--- program Path2 (robot UR5) ---
  Smooth(1)
  Set Ref.: Frame 2 at (-32.2, -480, 0) mm
  Set Tool: laser_fixture_tool
  Show laser_fixture_tool
  Set speed (1000.0 mm/s)
  MoveJ 1 to (-97.68, -19.69, 50.49) mm, rotated rx -95.37 ry 46.1 rz -97.44 deg; joints [-117.398, -152.62, -79.729, 61.497, 204.11, 54.589]
  MoveL 2 to (-97.68, -19.69, 50.49) mm, rotated rx -95.37 ry 46.1 rz -97.44 deg; joints [-117.398, -152.62, -79.729, 61.497, 204.11, 54.589]
  MoveL 3 to (1.91, -25.89, 44) mm, rotated rx -95.37 ry 46.1 rz -97.44 deg; joints [-108.024, -149.891, -88.195, 72.69, 194.926, 60.358]
  MoveL 4 to (1.91, -25.89, 44) mm, rotated rx -95.37 ry 46.1 rz -97.44 deg; joints [-108.024, -149.891, -88.195, 72.69, 194.926, 60.358]
  Set speed (100.0 mm/s)
  MoveL 5 to (1.98, -24.59, 43.9) mm, rotated rx -94.01 ry 38.49 rz -96.43 deg; joints [-108.115, -149.874, -89.181, 71.68, 194.519, 50.789]
  MoveL 6 to (2.06, -23.31, 43.74) mm, rotated rx -92.48 ry 28.02 rz -95.27 deg; joints [-108.188, -149.973, -90.447, 69.355, 194.248, 36.704]
  MoveL 7 to (2.12, -22.3, 43.59) mm, rotated rx -91.26 ry 16 rz -94.57 deg; joints [-108.24, -150.074, -91.694, 66.761, 194.073, 20.852]
  MoveL 8 to (2.19, -21.29, 43.41) mm, rotated rx -90.07 ry 0.97 rz -94.25 deg; joints [-108.275, -150.182, -93.079, 63.558, 194.03, 1.259]
  MoveL 9 to (2.26, -20.27, 43.2) mm, rotated rx -88.73 ry -16.32 rz -94.53 deg; joints [-108.287, -150.286, -94.55, 59.834, 194.17, -21.172]
  MoveL 10 to (2.33, -19.25, 42.96) mm, rotated rx -86.87 ry -33.13 rz -95.71 deg; joints [-108.274, -150.382, -96, 55.867, 194.507, -43.358]
  MoveL 11 to (2.41, -18.24, 42.7) mm, rotated rx -83.97 ry -47.18 rz -98.2 deg; joints [-108.236, -150.476, -97.37, 51.853, 195.027, -62.813]
  MoveL 12 to (2.5, -17.15, 42.4) mm, rotated rx -78.9 ry -58.66 rz -102.94 deg; joints [-108.162, -150.604, -98.668, 47.676, 195.795, -79.986]
  MoveL 13 to (2.6, -15.98, 42.05) mm, rotated rx -70.11 ry -67.29 rz -111.42 deg; joints [-108.046, -150.804, -99.778, 43.597, 196.83, -94.499]
  MoveL 14 to (2.71, -14.82, 41.67) mm, rotated rx -56.63 ry -72.85 rz -124.58 deg; joints [-107.893, -151.088, -100.576, 40.065, 198.034, -105.875]
  MoveL 15 to (2.81, -13.7, 41.29) mm, rotated rx -39.3 ry -75.67 rz -141.58 deg; joints [-107.714, -151.441, -101.097, 37.153, 199.307, -114.647]
  MoveL 16 to (2.92, -12.62, 40.89) mm, rotated rx -21.62 ry -76.38 rz -158.93 deg; joints [-107.516, -151.847, -101.404, 34.774, 200.599, -121.547]
  MoveL 17 to (3.02, -11.55, 40.47) mm, rotated rx -6.64 ry -75.69 rz -173.56 deg; joints [-107.294, -152.307, -101.552, 32.769, 201.93, -127.281]
  MoveL 18 to (3.14, -10.42, 40.01) mm, rotated rx 5.46 ry -74.12 rz 174.75 deg; joints [-107.034, -152.855, -101.524, 31.037, 203.383, -132.45]
  MoveL 19 to (3.26, -9.3, 39.53) mm, rotated rx 13.98 ry -72.1 rz 166.68 deg; joints [-106.75, -153.449, -101.357, 29.617, 204.857, -136.867]
  MoveL 20 to (3.38, -8.19, 39.02) mm, rotated rx 20.16 ry -69.89 rz 160.98 deg; joints [-106.442, -154.081, -101.056, 28.479, 206.349, -140.71]
  MoveL 21 to (3.5, -7.16, 38.53) mm, rotated rx 24.31 ry -67.77 rz 157.31 deg; joints [-106.138, -154.692, -100.702, 27.595, 207.742, -143.855]
  MoveL 22 to (3.62, -6.13, 38.01) mm, rotated rx 27.45 ry -65.69 rz 154.67 deg; joints [-105.824, -155.305, -100.283, 26.893, 209.104, -146.603]
  MoveL 23 to (3.74, -5.11, 37.48) mm, rotated rx 29.93 ry -63.69 rz 152.7 deg; joints [-105.508, -155.909, -99.812, 26.36, 210.414, -148.998]
  MoveL 24 to (3.87, -4.1, 36.93) mm, rotated rx 31.98 ry -61.8 rz 151.18 deg; joints [-105.197, -156.492, -99.304, 25.985, 211.65, -151.075]
  MoveL 25 to (3.99, -3.1, 36.36) mm, rotated rx 33.74 ry -60.04 rz 149.95 deg; joints [-104.899, -157.044, -98.773, 25.755, 212.794, -152.865]
  MoveL 26 to (4.12, -2.14, 35.78) mm, rotated rx 35.25 ry -58.46 rz 148.94 deg; joints [-104.624, -157.546, -98.249, 25.647, 213.814, -154.372]
  MoveL 27 to (4.25, -1.18, 35.18) mm, rotated rx 36.76 ry -56.98 rz 147.94 deg; joints [-104.37, -158.013, -97.693, 25.681, 214.733, -155.685]
  MoveL 28 to (4.37, -0.31, 34.6) mm, rotated rx 38.13 ry -55.7 rz 147.04 deg; joints [-104.155, -158.41, -97.17, 25.81, 215.493, -156.743]
  MoveL 29 to (4.5, 0.55, 34.01) mm, rotated rx 39.62 ry -54.47 rz 146.03 deg; joints [-103.959, -158.78, -96.605, 26.059, 216.174, -157.692]
  MoveL 30 to (4.62, 1.39, 33.4) mm, rotated rx 41.27 ry -53.25 rz 144.88 deg; joints [-103.782, -159.123, -95.99, 26.432, 216.78, -158.557]
  MoveL 31 to (4.74, 2.19, 32.8) mm, rotated rx 42.33 ry -52.31 rz 144.22 deg; joints [-103.635, -159.404, -95.553, 26.685, 217.275, -159.223]
  MoveL 32 to (4.91, 3.31, 31.9) mm, rotated rx 44.8 ry -50.73 rz 142.45 deg; joints [-103.451, -159.789, -94.649, 27.444, 217.892, -160.186]
  MoveL 33 to (5.08, 4.4, 30.96) mm, rotated rx 47.43 ry -49.14 rz 140.54 deg; joints [-103.305, -160.117, -93.707, 28.355, 218.378, -161.045]
  MoveL 34 to (5.25, 5.45, 29.99) mm, rotated rx 49.49 ry -47.83 rz 139.06 deg; joints [-103.198, -160.376, -92.96, 29.156, 218.736, -161.713]
  MoveL 35 to (5.43, 6.44, 28.99) mm, rotated rx 50.93 ry -46.84 rz 138.05 deg; joints [-103.118, -160.586, -92.43, 29.783, 218.999, -162.207]
  MoveL 36 to (5.61, 7.35, 28) mm, rotated rx 51.83 ry -46.14 rz 137.47 deg; joints [-103.051, -160.768, -92.087, 30.223, 219.211, -162.569]
  MoveL 37 to (5.8, 8.16, 27.05) mm, rotated rx 52.21 ry -45.7 rz 137.3 deg; joints [-102.985, -160.938, -91.909, 30.456, 219.407, -162.832]
  MoveL 38 to (6.01, 8.91, 26.1) mm, rotated rx 52.19 ry -45.41 rz 137.45 deg; joints [-102.907, -161.118, -91.833, 30.519, 219.628, -163.057]
  MoveL 39 to (6.25, 9.59, 25.16) mm, rotated rx 51.89 ry -45.19 rz 137.87 deg; joints [-102.804, -161.322, -91.806, 30.444, 219.904, -163.292]
  MoveL 40 to (6.49, 10.19, 24.25) mm, rotated rx 51.29 ry -45.01 rz 138.58 deg; joints [-102.671, -161.555, -91.827, 30.209, 220.257, -163.553]
  MoveL 41 to (6.77, 10.75, 23.33) mm, rotated rx 50.5 ry -44.77 rz 139.49 deg; joints [-102.494, -161.833, -91.835, 29.864, 220.718, -163.892]
  MoveL 42 to (7.09, 11.26, 22.39) mm, rotated rx 49.64 ry -44.4 rz 140.54 deg; joints [-102.268, -162.162, -91.794, 29.446, 221.298, -164.331]
  MoveL 43 to (7.44, 11.72, 21.44) mm, rotated rx 48.8 ry -43.88 rz 141.63 deg; joints [-101.995, -162.534, -91.675, 28.993, 221.99, -164.871]
  MoveL 44 to (7.81, 12.11, 20.53) mm, rotated rx 48.83 ry -43.04 rz 142.03 deg; joints [-101.733, -162.885, -91.275, 28.886, 222.626, -165.478]
  MoveL 45 to (7.95, 12.23, 20.22) mm, rotated rx 49.41 ry -42.62 rz 141.68 deg; joints [-101.675, -162.97, -90.985, 29.096, 222.751, -165.687]
  Set speed (1000.0 mm/s)
  MoveL 46 to (7.95, 12.23, 20.22) mm, rotated rx 49.41 ry -42.62 rz 141.68 deg; joints [-101.675, -162.97, -90.985, 29.096, 222.751, -165.687]
  MoveL 47 to (-73.7, -20.03, -27.66) mm, rotated rx 49.41 ry -42.62 rz 141.68 deg; joints [-108.268, -173.052, -72.375, 25.011, 227.608, -159.391]
  Set speed (1000.0 mm/s)
  MoveL 48 to (-97.55, 35.36, 42.52) mm, rotated rx -88.89 ry -10.51 rz -96.06 deg; joints [-120.475, -150.967, -92.517, 60.869, 204.643, -12.887]
  MoveL 49 to (1.91, 25.16, 44.42) mm, rotated rx -88.89 ry -10.51 rz -96.06 deg; joints [-110.164, -147.723, -102.71, 66.031, 194.349, -14.776]
  MoveL 50 to (1.91, 25.16, 44.42) mm, rotated rx -88.89 ry -10.51 rz -96.06 deg; joints [-110.164, -147.723, -102.71, 66.031, 194.349, -14.776]
  Set speed (100.0 mm/s)
  MoveL 51 to (1.98, 25.72, 43.25) mm, rotated rx -88.19 ry -17.29 rz -96.08 deg; joints [-110.132, -148.034, -103.098, 64.289, 194.692, -23.923]
  MoveL 52 to (2.06, 26.23, 42.05) mm, rotated rx -87.4 ry -25.95 rz -95.93 deg; joints [-110.04, -148.436, -103.065, 62.671, 195.424, -34.491]
  MoveL 53 to (2.12, 26.6, 41.1) mm, rotated rx -86.33 ry -36.31 rz -96.18 deg; joints [-109.931, -148.826, -102.954, 61.128, 196.192, -46.606]
  MoveL 54 to (2.19, 26.95, 40.14) mm, rotated rx -84.48 ry -49.54 rz -97.24 deg; joints [-109.789, -149.268, -102.655, 59.677, 197.122, -61.387]
  MoveL 55 to (2.26, 27.27, 39.15) mm, rotated rx -79.85 ry -65.51 rz -101.13 deg; joints [-109.61, -149.762, -102.145, 58.387, 198.206, -78.71]
  MoveL 56 to (2.33, 27.58, 38.15) mm, rotated rx -55.43 ry -81.59 rz -124.86 deg; joints [-109.399, -150.29, -101.463, 57.275, 199.392, -96.746]
  MoveL 57 to (2.41, 27.86, 37.15) mm, rotated rx 58.45 ry -79.77 rz 121.96 deg; joints [-109.16, -150.846, -100.674, 56.248, 200.649, -113.072]
  MoveL 58 to (2.5, 28.14, 36.05) mm, rotated rx 74.81 ry -66.9 rz 106.44 deg; joints [-108.873, -151.466, -99.702, 55.284, 202.062, -127.151]
  MoveL 59 to (2.6, 28.42, 34.87) mm, rotated rx 78.42 ry -56.07 rz 103.87 deg; joints [-108.537, -152.135, -98.547, 54.435, 203.605, -138.342]
  MoveL 60 to (2.71, 28.68, 33.67) mm, rotated rx 79.75 ry -47.86 rz 103.7 deg; joints [-108.18, -152.789, -97.305, 53.779, 205.14, -146.526]
  MoveL 61 to (2.81, 28.9, 32.51) mm, rotated rx 80.34 ry -41.76 rz 104.33 deg; joints [-107.819, -153.406, -96.068, 53.252, 206.603, -152.411]
  MoveL 62 to (2.92, 29.1, 31.38) mm, rotated rx 80.63 ry -37.16 rz 105.29 deg; joints [-107.46, -153.987, -94.871, 52.799, 207.986, -156.733]
  MoveL 63 to (3.02, 29.28, 30.24) mm, rotated rx 80.77 ry -33.45 rz 106.42 deg; joints [-107.092, -154.551, -93.682, 52.386, 209.335, -160.107]
  MoveL 64 to (3.14, 29.44, 29.03) mm, rotated rx 80.98 ry -29.94 rz 107.64 deg; joints [-106.696, -155.114, -92.391, 52.087, 210.724, -163.092]
  MoveL 65 to (3.26, 29.58, 27.82) mm, rotated rx 81.2 ry -26.87 rz 108.91 deg; joints [-106.294, -155.65, -91.099, 51.853, 212.077, -165.555]
  MoveL 66 to (3.38, 29.7, 26.61) mm, rotated rx 81.49 ry -24.03 rz 110.17 deg; joints [-105.888, -156.149, -89.791, 51.726, 213.39, -167.677]
  MoveL 67 to (3.5, 29.79, 25.46) mm, rotated rx 81.76 ry -21.7 rz 111.4 deg; joints [-105.504, -156.6, -88.587, 51.615, 214.592, -169.337]
  MoveL 68 to (3.62, 29.86, 24.31) mm, rotated rx 82.05 ry -19.58 rz 112.61 deg; joints [-105.124, -157.021, -87.412, 51.55, 215.741, -170.757]
  MoveL 69 to (3.74, 29.91, 23.17) mm, rotated rx 82.39 ry -17.66 rz 113.77 deg; joints [-104.756, -157.407, -86.281, 51.538, 216.822, -171.975]
  MoveL 70 to (3.87, 29.93, 22.02) mm, rotated rx 82.78 ry -15.88 rz 114.85 deg; joints [-104.406, -157.754, -85.205, 51.582, 217.821, -173.027]
  MoveL 71 to (3.99, 29.93, 20.87) mm, rotated rx 83.21 ry -14.24 rz 115.84 deg; joints [-104.082, -158.056, -84.199, 51.692, 218.723, -173.941]
  MoveL 72 to (4.12, 29.91, 19.74) mm, rotated rx 83.63 ry -12.81 rz 116.73 deg; joints [-103.789, -158.322, -83.295, 51.823, 219.514, -174.697]
  MoveL 73 to (4.25, 29.87, 18.61) mm, rotated rx 84.14 ry -11.38 rz 117.48 deg; joints [-103.53, -158.531, -82.452, 52.062, 220.197, -175.401]
  MoveL 74 to (4.37, 29.81, 17.57) mm, rotated rx 84.59 ry -10.22 rz 118.11 deg; joints [-103.314, -158.707, -81.751, 52.28, 220.752, -175.949]
  MoveL 75 to (4.5, 29.73, 16.53) mm, rotated rx 85.11 ry -9.02 rz 118.63 deg; joints [-103.127, -158.835, -81.096, 52.592, 221.22, -176.485]
  MoveL 76 to (4.62, 29.62, 15.5) mm, rotated rx 85.75 ry -7.69 rz 119.02 deg; joints [-102.972, -158.905, -80.479, 53.039, 221.596, -177.042]
  MoveL 77 to (4.74, 29.5, 14.5) mm, rotated rx 85.8 ry -7.44 rz 119.58 deg; joints [-102.802, -159.131, -80.043, 52.942, 222.007, -177.183]
  MoveL 78 to (4.91, 29.28, 13.09) mm, rotated rx 86.75 ry -5.66 rz 119.88 deg; joints [-102.658, -159.144, -79.34, 53.684, 222.322, -177.88]
  MoveL 79 to (5.08, 29.01, 11.67) mm, rotated rx 87.98 ry -3.51 rz 119.97 deg; joints [-102.577, -159.024, -78.704, 54.74, 222.463, -178.695]
  MoveL 80 to (5.25, 28.69, 10.28) mm, rotated rx 89.05 ry -1.64 rz 120.03 deg; joints [-102.522, -158.914, -78.188, 55.701, 222.53, -179.393]
  MoveL 81 to (5.43, 28.33, 8.92) mm, rotated rx 89.88 ry -0.2 rz 120.1 deg; joints [-102.475, -158.856, -77.771, 56.457, 222.571, -179.927]
  MoveL 82 to (5.61, 27.93, 7.64) mm, rotated rx 90.48 ry 0.83 rz 120.2 deg; joints [-102.423, -158.862, -77.418, 56.992, 222.62, -180.305]
  MoveL 83 to (5.8, 27.51, 6.46) mm, rotated rx 90.82 ry 1.4 rz 120.38 deg; joints [-102.35, -158.951, -77.096, 57.254, 222.721, -180.511]
  MoveL 84 to (6.01, 27.06, 5.34) mm, rotated rx 90.99 ry 1.67 rz 120.66 deg; joints [-102.25, -159.104, -76.764, 57.323, 222.886, -180.606]
  MoveL 85 to (6.25, 26.58, 4.28) mm, rotated rx 91.07 ry 1.79 rz 121.02 deg; joints [-102.12, -159.301, -76.395, 57.266, 223.122, -180.64]
  MoveL 86 to (6.49, 26.1, 3.3) mm, rotated rx 91.01 ry 1.65 rz 121.54 deg; joints [-101.946, -159.565, -75.976, 57.014, 223.47, -180.583]
  MoveL 87 to (6.77, 25.58, 2.36) mm, rotated rx 90.92 ry 1.46 rz 122.22 deg; joints [-101.725, -159.869, -75.473, 56.67, 223.927, -180.506]
  MoveL 88 to (7.09, 25.02, 1.44) mm, rotated rx 90.84 ry 1.3 rz 123.04 deg; joints [-101.459, -160.198, -74.88, 56.28, 224.49, -180.438]
  MoveL 89 to (7.44, 24.43, 0.58) mm, rotated rx 90.81 ry 1.21 rz 124 deg; joints [-101.151, -160.532, -74.203, 55.884, 225.142, -180.397]
  MoveL 90 to (7.81, 23.83, -0.22) mm, rotated rx 91.3 ry 1.88 rz 124.66 deg; joints [-100.929, -160.632, -73.599, 56.053, 225.559, -180.608]
  MoveL 91 to (7.95, 23.62, -0.48) mm, rotated rx 91.81 ry 2.62 rz 124.61 deg; joints [-100.934, -160.496, -73.485, 56.516, 225.491, -180.847]
  Set speed (1000.0 mm/s)
  MoveL 92 to (7.95, 23.62, -0.48) mm, rotated rx 91.81 ry 2.62 rz 124.61 deg; joints [-100.934, -160.496, -73.485, 56.516, 225.491, -180.847]
  MoveL 93 to (-74.39, -33.03, 2.67) mm, rotated rx 91.81 ry 2.62 rz 124.61 deg; joints [-106.621, -168.974, -51.295, 42.589, 231.173, -181.169]
  Set speed (1000.0 mm/s)
  MoveL 94 to (-97.68, 53.58, -8.19) mm, rotated rx -72.98 ry -72.89 rz -107.76 deg; joints [-120.487, -158.48, -90.615, 58.994, 209.415, -82.414]
  MoveL 95 to (1.91, 51.05, 0.42) mm, rotated rx -72.98 ry -72.89 rz -107.76 deg; joints [-110.485, -154.518, -103.068, 62.737, 199.64, -87.613]
  MoveL 96 to (1.91, 51.05, 0.42) mm, rotated rx -72.98 ry -72.89 rz -107.76 deg; joints [-110.485, -154.518, -103.068, 62.737, 199.64, -87.613]
  Set speed (100.0 mm/s)
  MoveL 97 to (1.98, 50.31, -0.65) mm, rotated rx -60.07 ry -79.99 rz -120.31 deg; joints [-110.333, -154.806, -102.376, 62.619, 200.171, -95.008]
  MoveL 98 to (2.06, 49.53, -1.69) mm, rotated rx 22.06 ry -84.98 rz 158.02 deg; joints [-110.154, -155.029, -101.323, 63.16, 200.811, -104.247]
  MoveL 99 to (2.12, 48.9, -2.48) mm, rotated rx 72.87 ry -75.39 rz 107.66 deg; joints [-109.98, -155.191, -100.295, 63.767, 201.447, -114.914]
  MoveL 100 to (2.19, 48.24, -3.26) mm, rotated rx 82.4 ry -60.69 rz 98.7 deg; joints [-109.787, -155.315, -99.138, 64.567, 202.148, -128.264]
  MoveL 101 to (2.26, 47.54, -4.04) mm, rotated rx 85.87 ry -43.48 rz 95.99 deg; joints [-109.575, -155.395, -97.868, 65.545, 202.908, -143.564]
  MoveL 102 to (2.33, 46.83, -4.81) mm, rotated rx 87.6 ry -26.64 rz 95.35 deg; joints [-109.346, -155.428, -96.545, 66.622, 203.71, -158.244]
  MoveL 103 to (2.41, 46.1, -5.55) mm, rotated rx 88.77 ry -12.46 rz 95.7 deg; joints [-109.101, -155.424, -95.197, 67.721, 204.559, -170.17]
  MoveL 104 to (2.5, 45.3, -6.35) mm, rotated rx 89.92 ry -0.69 rz 96.69 deg; joints [-108.819, -155.373, -93.741, 68.926, 205.509, -179.481]
  MoveL 105 to (2.6, 44.41, -7.18) mm, rotated rx 91.24 ry 8.62 rz 98.2 deg; joints [-108.504, -155.267, -92.215, 70.221, 206.544, -186.174]
  MoveL 106 to (2.71, 43.5, -8) mm, rotated rx 92.7 ry 15.52 rz 100 deg; joints [-108.181, -155.111, -90.759, 71.5, 207.574, -190.539]
  MoveL 107 to (2.81, 42.61, -8.78) mm, rotated rx 94.25 ry 20.57 rz 101.95 deg; joints [-107.86, -154.925, -89.421, 72.692, 208.569, -193.276]
  MoveL 108 to (2.92, 41.72, -9.51) mm, rotated rx 95.86 ry 24.37 rz 103.96 deg; joints [-107.544, -154.719, -88.201, 73.792, 209.522, -194.995]
  MoveL 109 to (3.02, 40.83, -10.23) mm, rotated rx 97.55 ry 27.42 rz 106.06 deg; joints [-107.224, -154.491, -87.054, 74.845, 210.466, -196.106]
  MoveL 110 to (3.14, 39.86, -10.98) mm, rotated rx 99.48 ry 30.17 rz 108.37 deg; joints [-106.885, -154.21, -85.922, 75.969, 211.439, -196.911]
  MoveL 111 to (3.26, 38.88, -11.71) mm, rotated rx 101.51 ry 32.49 rz 110.76 deg; joints [-106.544, -153.899, -84.869, 77.078, 212.397, -197.407]
  MoveL 112 to (3.38, 37.89, -12.42) mm, rotated rx 103.67 ry 34.51 rz 113.24 deg; joints [-106.203, -153.549, -83.898, 78.205, 213.333, -197.712]
  MoveL 113 to (3.5, 36.94, -13.07) mm, rotated rx 105.76 ry 36.1 rz 115.6 deg; joints [-105.88, -153.203, -83.052, 79.239, 214.203, -197.823]
  MoveL 114 to (3.62, 35.99, -13.7) mm, rotated rx 107.89 ry 37.46 rz 117.96 deg; joints [-105.562, -152.84, -82.283, 80.256, 215.042, -197.829]
  MoveL 115 to (3.74, 35.01, -14.32) mm, rotated rx 110.03 ry 38.63 rz 120.28 deg; joints [-105.254, -152.466, -81.597, 81.254, 215.836, -197.771]
  MoveL 116 to (3.87, 34.03, -14.91) mm, rotated rx 112.14 ry 39.64 rz 122.52 deg; joints [-104.962, -152.088, -80.998, 82.233, 216.568, -197.681]
  MoveL 117 to (3.99, 33.04, -15.49) mm, rotated rx 114.19 ry 40.52 rz 124.65 deg; joints [-104.693, -151.712, -80.486, 83.185, 217.226, -197.584]
  MoveL 118 to (4.12, 32.05, -16.04) mm, rotated rx 116.12 ry 41.29 rz 126.61 deg; joints [-104.452, -151.356, -80.062, 84.085, 217.793, -197.494]
  MoveL 119 to (4.25, 31.06, -16.56) mm, rotated rx 118.01 ry 42.05 rz 128.46 deg; joints [-104.243, -150.995, -79.727, 84.999, 218.263, -197.458]
  MoveL 120 to (4.37, 30.12, -17.03) mm, rotated rx 119.71 ry 42.73 rz 130.07 deg; joints [-104.077, -150.667, -79.485, 85.842, 218.616, -197.464]
  MoveL 121 to (4.5, 29.18, -17.48) mm, rotated rx 121.44 ry 43.48 rz 131.62 deg; joints [-103.941, -150.324, -79.322, 86.736, 218.878, -197.545]
  MoveL 122 to (4.62, 28.23, -17.9) mm, rotated rx 123.23 ry 44.32 rz 133.16 deg; joints [-103.84, -149.961, -79.242, 87.702, 219.042, -197.713]
  MoveL 123 to (4.74, 27.31, -18.29) mm, rotated rx 124.62 ry 44.85 rz 134.39 deg; joints [-103.737, -149.704, -79.122, 88.405, 219.214, -197.761]
  MoveL 124 to (4.91, 25.97, -18.81) mm, rotated rx 127.16 ry 46.15 rz 136.42 deg; joints [-103.679, -149.19, -79.191, 89.834, 219.202, -198.177]
  MoveL 125 to (5.08, 24.62, -19.29) mm, rotated rx 129.83 ry 47.58 rz 138.48 deg; joints [-103.675, -148.665, -79.374, 91.349, 219.034, -198.729]
  MoveL 126 to (5.25, 23.24, -19.71) mm, rotated rx 132.09 ry 48.72 rz 140.24 deg; joints [-103.675, -148.262, -79.507, 92.588, 218.852, -199.185]
  MoveL 127 to (5.43, 21.89, -20.07) mm, rotated rx 133.83 ry 49.53 rz 141.6 deg; joints [-103.661, -147.994, -79.546, 93.49, 218.711, -199.492]
  MoveL 128 to (5.61, 20.58, -20.37) mm, rotated rx 135.07 ry 50.01 rz 142.61 deg; joints [-103.622, -147.835, -79.488, 94.089, 218.641, -199.638]
  MoveL 129 to (5.8, 19.35, -20.59) mm, rotated rx 135.83 ry 50.18 rz 143.27 deg; joints [-103.551, -147.767, -79.328, 94.4, 218.675, -199.606]
  MoveL 130 to (6.01, 18.15, -20.76) mm, rotated rx 136.28 ry 50.1 rz 143.73 deg; joints [-103.442, -147.751, -79.081, 94.521, 218.817, -199.415]
  MoveL 131 to (6.25, 17, -20.88) mm, rotated rx 136.57 ry 49.83 rz 144.12 deg; joints [-103.296, -147.749, -78.771, 94.534, 219.066, -199.092]
  MoveL 132 to (6.49, 15.91, -20.95) mm, rotated rx 136.73 ry 49.35 rz 144.46 deg; joints [-103.105, -147.757, -78.393, 94.436, 219.449, -198.619]
  MoveL 133 to (6.77, 14.83, -20.97) mm, rotated rx 136.92 ry 48.72 rz 144.9 deg; joints [-102.867, -147.739, -77.968, 94.322, 219.957, -198.032]
  MoveL 134 to (7.09, 13.76, -20.94) mm, rotated rx 137.25 ry 48 rz 145.51 deg; joints [-102.585, -147.671, -77.519, 94.247, 220.579, -197.361]
  MoveL 135 to (7.44, 12.71, -20.87) mm, rotated rx 137.77 ry 47.23 rz 146.33 deg; joints [-102.266, -147.538, -77.077, 94.258, 221.294, -196.645]
  MoveL 136 to (7.81, 11.72, -20.75) mm, rotated rx 138.98 ry 46.94 rz 147.56 deg; joints [-102.021, -147.228, -76.896, 94.747, 221.787, -196.225]
  MoveL 137 to (7.95, 11.39, -20.7) mm, rotated rx 139.78 ry 47.2 rz 148.18 deg; joints [-102.006, -147.032, -77.006, 95.203, 221.761, -196.298]
  Set speed (1000.0 mm/s)
  MoveL 138 to (7.95, 11.39, -20.7) mm, rotated rx 139.78 ry 47.2 rz 148.18 deg; joints [-102.006, -147.032, -77.006, 95.203, 221.761, -196.298]
  MoveL 139 to (-73.7, -13.94, 31.18) mm, rotated rx 139.78 ry 47.2 rz 148.18 deg; joints [-108.931, -148.976, -64.289, 79.063, 226.36, -203.756]
  Set speed (1000.0 mm/s)
  MoveL 140 to (-97.68, 19.69, -50.49) mm, rotated rx 84.63 ry -46.1 rz 97.44 deg; joints [-117.798, -165.768, -78.334, 56.973, 211.556, -139.855]
  MoveL 141 to (1.91, 25.89, -44) mm, rotated rx 84.63 ry -46.1 rz 97.44 deg; joints [-108.738, -161.585, -91.609, 63.461, 202.592, -142.771]
  MoveL 142 to (1.91, 25.89, -44) mm, rotated rx 84.63 ry -46.1 rz 97.44 deg; joints [-108.738, -161.585, -91.609, 63.461, 202.592, -142.771]
  Set speed (100.0 mm/s)
  MoveL 143 to (1.98, 24.59, -43.9) mm, rotated rx 85.99 ry -38.49 rz 96.43 deg; joints [-108.636, -161.508, -90.877, 64.247, 202.775, -148.954]
  MoveL 144 to (2.06, 23.31, -43.74) mm, rotated rx 87.52 ry -28.02 rz 95.27 deg; joints [-108.573, -161.275, -90.128, 65.736, 202.779, -157.189]
  MoveL 145 to (2.12, 22.3, -43.59) mm, rotated rx 88.74 ry -16 rz 94.57 deg; joints [-108.525, -161.003, -89.455, 67.324, 202.774, -166.881]
  MoveL 146 to (2.19, 21.29, -43.41) mm, rotated rx 89.93 ry -0.97 rz 94.25 deg; joints [-108.485, -160.649, -88.774, 69.236, 202.73, -179.201]
  MoveL 147 to (2.26, 20.27, -43.2) mm, rotated rx 91.27 ry 16.32 rz 94.53 deg; joints [-108.451, -160.202, -88.099, 71.478, 202.652, -193.389]
  MoveL 148 to (2.33, 19.25, -42.96) mm, rotated rx 93.13 ry 33.13 rz 95.71 deg; joints [-108.419, -159.674, -87.452, 73.968, 202.564, -206.849]
  MoveL 149 to (2.41, 18.24, -42.7) mm, rotated rx 96.03 ry 47.18 rz 98.2 deg; joints [-108.381, -159.07, -86.83, 76.657, 202.504, -217.387]
  MoveL 150 to (2.5, 17.15, -42.4) mm, rotated rx 101.1 ry 58.66 rz 102.94 deg; joints [-108.333, -158.333, -86.216, 79.744, 202.471, -225.046]
  MoveL 151 to (2.6, 15.98, -42.05) mm, rotated rx 109.89 ry 67.29 rz 111.42 deg; joints [-108.273, -157.452, -85.651, 83.202, 202.477, -229.833]
  MoveL 152 to (2.71, 14.82, -41.67) mm, rotated rx 123.37 ry 72.85 rz 124.58 deg; joints [-108.204, -156.491, -85.203, 86.74, 202.53, -232.203]
  MoveL 153 to (2.81, 13.7, -41.29) mm, rotated rx 140.7 ry 75.67 rz 141.58 deg; joints [-108.123, -155.493, -84.879, 90.193, 202.644, -232.933]
  MoveL 154 to (2.92, 12.62, -40.89) mm, rotated rx 158.38 ry 76.38 rz 158.93 deg; joints [-108.032, -154.475, -84.671, 93.513, 202.818, -232.673]
  MoveL 155 to (3.02, 11.55, -40.47) mm, rotated rx 173.36 ry 75.69 rz 173.56 deg; joints [-107.928, -153.412, -84.567, 96.798, 203.051, -231.796]
  MoveL 156 to (3.14, 10.42, -40.01) mm, rotated rx -174.54 ry 74.12 rz -174.75 deg; joints [-107.81, -152.234, -84.589, 100.273, 203.333, -230.532]
  MoveL 157 to (3.26, 9.3, -39.53) mm, rotated rx -166.02 ry 72.1 rz -166.68 deg; joints [-107.682, -151.008, -84.733, 103.723, 203.666, -228.989]
  MoveL 158 to (3.38, 8.19, -39.02) mm, rotated rx -159.84 ry 69.89 rz -160.98 deg; joints [-107.546, -149.736, -85.005, 107.166, 204.034, -227.306]
  MoveL 159 to (3.5, 7.16, -38.53) mm, rotated rx -155.69 ry 67.77 rz -157.31 deg; joints [-107.406, -148.512, -85.355, 110.345, 204.433, -225.591]
  MoveL 160 to (3.62, 6.13, -38.01) mm, rotated rx -152.55 ry 65.69 rz -154.67 deg; joints [-107.258, -147.285, -85.789, 113.432, 204.86, -223.86]
  MoveL 161 to (3.74, 5.11, -37.48) mm, rotated rx -150.07 ry 63.69 rz -152.7 deg; joints [-107.108, -146.075, -86.289, 116.393, 205.297, -222.176]
  MoveL 162 to (3.87, 4.1, -36.93) mm, rotated rx -148.02 ry 61.8 rz -151.18 deg; joints [-106.96, -144.907, -86.837, 119.2, 205.723, -220.594]
  MoveL 163 to (3.99, 3.1, -36.36) mm, rotated rx -146.26 ry 60.04 rz -149.95 deg; joints [-106.818, -143.804, -87.409, 121.823, 206.12, -219.155]
  MoveL 164 to (4.12, 2.14, -35.78) mm, rotated rx -144.75 ry 58.46 rz -148.94 deg; joints [-106.687, -142.798, -87.972, 124.201, 206.47, -217.89]
  MoveL 165 to (4.25, 1.18, -35.18) mm, rotated rx -143.24 ry 56.98 rz -147.94 deg; joints [-106.574, -141.87, -88.543, 126.441, 206.739, -216.823]
  MoveL 166 to (4.37, 0.31, -34.6) mm, rotated rx -141.87 ry 55.7 rz -147.04 deg; joints [-106.486, -141.086, -89.061, 128.382, 206.922, -215.987]
  MoveL 167 to (4.5, -0.55, -34.01) mm, rotated rx -140.38 ry 54.47 rz -146.03 deg; joints [-106.422, -140.363, -89.588, 130.269, 207.008, -215.324]
  MoveL 168 to (4.62, -1.39, -33.4) mm, rotated rx -138.73 ry 53.25 rz -144.88 deg; joints [-106.384, -139.699, -90.125, 132.139, 206.985, -214.832]
  MoveL 169 to (4.74, -2.19, -32.8) mm, rotated rx -137.67 ry 52.31 rz -144.22 deg; joints [-106.33, -139.146, -90.533, 133.59, 207.037, -214.312]
  MoveL 170 to (4.91, -3.31, -31.9) mm, rotated rx -135.2 ry 50.73 rz -142.45 deg; joints [-106.34, -138.411, -91.245, 136.022, 206.747, -214.02]
  MoveL 171 to (5.08, -4.4, -30.96) mm, rotated rx -132.57 ry 49.14 rz -140.54 deg; joints [-106.392, -137.79, -91.937, 138.413, 206.276, -213.961]
  MoveL 172 to (5.25, -5.45, -29.99) mm, rotated rx -130.51 ry 47.83 rz -139.06 deg; joints [-106.432, -137.302, -92.468, 140.351, 205.855, -213.905]
  MoveL 173 to (5.43, -6.44, -28.99) mm, rotated rx -129.07 ry 46.84 rz -138.05 deg; joints [-106.446, -136.918, -92.837, 141.797, 205.552, -213.79]
  MoveL 174 to (5.61, -7.35, -28) mm, rotated rx -128.17 ry 46.14 rz -137.47 deg; joints [-106.429, -136.595, -93.083, 142.83, 205.392, -213.581]
  MoveL 175 to (5.8, -8.16, -27.05) mm, rotated rx -127.79 ry 45.7 rz -137.3 deg; joints [-106.376, -136.294, -93.238, 143.512, 205.405, -213.232]
  MoveL 176 to (6.01, -8.91, -26.1) mm, rotated rx -127.81 ry 45.41 rz -137.45 deg; joints [-106.288, -135.968, -93.357, 144.008, 205.581, -212.718]
  MoveL 177 to (6.25, -9.59, -25.16) mm, rotated rx -128.11 ry 45.19 rz -137.87 deg; joints [-106.166, -135.58, -93.489, 144.453, 205.902, -212.032]
  MoveL 178 to (6.49, -10.19, -24.25) mm, rotated rx -128.71 ry 45.01 rz -138.58 deg; joints [-106.005, -135.114, -93.646, 144.863, 206.402, -211.144]
  MoveL 179 to (6.77, -10.75, -23.33) mm, rotated rx -129.5 ry 44.77 rz -139.49 deg; joints [-105.803, -134.53, -93.879, 145.384, 207.06, -210.055]
  MoveL 180 to (7.09, -11.26, -22.39) mm, rotated rx -130.36 ry 44.4 rz -140.54 deg; joints [-105.562, -133.816, -94.215, 146.085, 207.857, -208.791]
  MoveL 181 to (7.44, -11.72, -21.44) mm, rotated rx -131.2 ry 43.88 rz -141.63 deg; joints [-105.288, -132.981, -94.67, 146.997, 208.765, -207.409]
  MoveL 182 to (7.81, -12.11, -20.53) mm, rotated rx -131.17 ry 43.04 rz -142.03 deg; joints [-105.089, -132.15, -95.302, 148.426, 209.348, -206.329]
  MoveL 183 to (7.95, -12.23, -20.22) mm, rotated rx -130.59 ry 42.62 rz -141.68 deg; joints [-105.089, -131.924, -95.584, 149.185, 209.271, -206.201]
  Set speed (1000.0 mm/s)
  MoveL 184 to (7.95, -12.23, -20.22) mm, rotated rx -130.59 ry 42.62 rz -141.68 deg; joints [-105.089, -131.924, -95.584, 149.185, 209.271, -206.201]
  MoveL 185 to (-73.7, 20.03, 27.66) mm, rotated rx -130.59 ry 42.62 rz -141.68 deg; joints [-115.878, -132.254, -91.544, 125.938, 208.905, -228.491]
  Set speed (1000.0 mm/s)
  MoveL 186 to (-97.68, -33.88, -42.3) mm, rotated rx 91.25 ry 13.6 rz 95.3 deg; joints [-115.325, -167.015, -66.464, 55.883, 210.352, -191.529]
  MoveL 187 to (1.91, -25.16, -44.42) mm, rotated rx 91.25 ry 13.6 rz 95.3 deg; joints [-106.938, -162.85, -79.387, 65.483, 201.975, -190.592]
  MoveL 188 to (1.91, -25.16, -44.42) mm, rotated rx 91.25 ry 13.6 rz 95.3 deg; joints [-106.938, -162.85, -79.387, 65.483, 201.975, -190.592]
  Set speed (100.0 mm/s)
  MoveL 189 to (1.98, -25.72, -43.25) mm, rotated rx 91.96 ry 21.25 rz 95.4 deg; joints [-106.959, -162.497, -79.273, 66.717, 201.72, -196.665]
  MoveL 190 to (2.06, -26.23, -42.05) mm, rotated rx 92.89 ry 31.77 rz 95.48 deg; joints [-107.04, -162.038, -79.441, 68.305, 201.13, -205.427]
  MoveL 191 to (2.12, -26.6, -41.1) mm, rotated rx 94.22 ry 43.79 rz 96.08 deg; joints [-107.13, -161.595, -79.652, 69.965, 200.51, -215.69]
  MoveL 192 to (2.19, -26.95, -40.14) mm, rotated rx 97.03 ry 58.77 rz 98.21 deg; joints [-107.24, -161.102, -79.959, 71.885, 199.753, -228.756]
  MoveL 193 to (2.26, -27.27, -39.15) mm, rotated rx 107.34 ry 75.7 rz 107.86 deg; joints [-107.368, -160.56, -80.358, 74.085, 198.856, -243.845]
  MoveL 194 to (2.33, -27.58, -38.15) mm, rotated rx -145.62 ry 84.21 rz -145.76 deg; joints [-107.505, -159.987, -80.813, 76.54, 197.862, -258.258]
  MoveL 195 to (2.41, -27.86, -37.15) mm, rotated rx -107.11 ry 71.69 rz -107.97 deg; joints [-107.643, -159.381, -81.279, 79.311, 196.804, -269.648]
  MoveL 196 to (2.5, -28.14, -36.05) mm, rotated rx -101.72 ry 60.01 rz -103.48 deg; joints [-107.789, -158.697, -81.783, 82.664, 195.608, -278.032]
  MoveL 197 to (2.6, -28.42, -34.87) mm, rotated rx -99.98 ry 50.58 rz -102.83 deg; joints [-107.937, -157.93, -82.3, 86.697, 194.292, -283.235]
  MoveL 198 to (2.71, -28.68, -33.67) mm, rotated rx -99.26 ry 43.47 rz -103.33 deg; joints [-108.07, -157.122, -82.767, 91.224, 192.979, -285.471]
  MoveL 199 to (2.81, -28.9, -32.51) mm, rotated rx -98.93 ry 38.14 rz -104.27 deg; joints [-108.181, -156.266, -83.149, 96.237, 191.749, -285.277]
  MoveL 200 to (2.92, -29.1, -31.38) mm, rotated rx -98.74 ry 34 rz -105.37 deg; joints [-108.27, -155.322, -83.459, 101.828, 190.634, -283.133]
  MoveL 201 to (3.02, -29.28, -30.24) mm, rotated rx -98.6 ry 30.56 rz -106.57 deg; joints [-108.34, -154.191, -83.759, 108.345, 189.624, -279.157]
  MoveL 202 to (3.14, -29.44, -29.03) mm, rotated rx -98.42 ry 27.34 rz -107.86 deg; joints [-108.396, -152.705, -84.185, 116.448, 188.676, -273.14]
  MoveL 203 to (3.26, -29.58, -27.82) mm, rotated rx -98.21 ry 24.49 rz -109.18 deg; joints [-108.432, -150.768, -84.91, 126.116, 187.923, -265.027]
  MoveL 204 to (3.38, -29.7, -26.61) mm, rotated rx -97.93 ry 21.87 rz -110.5 deg; joints [-108.448, -148.27, -86.216, 137.45, 187.412, -255.036]
  MoveL 205 to (3.5, -29.79, -25.46) mm, rotated rx -97.65 ry 19.66 rz -111.76 deg; joints [-108.442, -145.409, -88.187, 149.351, 187.236, -244.376]
  MoveL 206 to (3.62, -29.86, -24.31) mm, rotated rx -97.33 ry 17.64 rz -112.99 deg; joints [-108.419, -142.311, -90.831, 161.557, 187.359, -233.663]
  MoveL 207 to (3.74, -29.91, -23.17) mm, rotated rx -96.96 ry 15.79 rz -114.16 deg; joints [-108.379, -139.311, -93.855, 173.134, 187.737, -223.902]
  MoveL 208 to (3.87, -29.93, -22.02) mm, rotated rx -96.55 ry 14.08 rz -115.27 deg; joints [-108.326, -136.659, -96.907, 183.46, 188.295, -215.636]
  MoveL 209 to (3.99, -29.93, -20.87) mm, rotated rx -96.1 ry 12.51 rz -116.28 deg; joints [-108.263, -134.452, -99.745, 192.33, 188.95, -208.939]
  MoveL 210 to (4.12, -29.91, -19.74) mm, rotated rx -95.64 ry 11.09 rz -117.17 deg; joints [-108.195, -132.699, -102.223, 199.696, 189.626, -203.699]
  MoveL 211 to (4.25, -29.87, -18.61) mm, rotated rx -95.11 ry 9.71 rz -117.94 deg; joints [-108.128, -131.278, -104.43, 206.159, 190.262, -199.404]
  MoveL 212 to (4.37, -29.81, -17.57) mm, rotated rx -94.59 ry 8.48 rz -118.56 deg; joints [-108.068, -130.21, -106.242, 211.463, 190.802, -196.087]
  MoveL 213 to (4.5, -29.73, -16.53) mm, rotated rx -94 ry 7.22 rz -119.07 deg; joints [-108.013, -129.322, -107.91, 216.501, 191.263, -193.128]
  MoveL 214 to (4.62, -29.62, -15.5) mm, rotated rx -93.32 ry 5.89 rz -119.47 deg; joints [-107.966, -128.588, -109.478, 221.479, 191.636, -190.365]
  MoveL 215 to (4.74, -29.5, -14.5) mm, rotated rx -92.83 ry 4.94 rz -119.86 deg; joints [-107.918, -128.046, -110.663, 225.053, 192.025, -188.421]
  MoveL 216 to (4.91, -29.28, -13.09) mm, rotated rx -91.76 ry 3.03 rz -120.17 deg; joints [-107.876, -127.415, -112.524, 231.666, 192.324, -185.049]
  MoveL 217 to (5.08, -29.01, -11.67) mm, rotated rx -90.61 ry 1.04 rz -120.34 deg; joints [-107.848, -127.01, -114.261, 238.469, 192.495, -181.7]
  MoveL 218 to (5.25, -28.69, -10.28) mm, rotated rx -89.65 ry -0.59 rz -120.47 deg; joints [-107.824, -126.778, -115.618, 243.991, 192.649, -179.038]
  MoveL 219 to (5.43, -28.33, -8.92) mm, rotated rx -88.94 ry -1.79 rz -120.6 deg; joints [-107.801, -126.627, -116.608, 248.005, 192.805, -177.136]
  MoveL 220 to (5.61, -27.93, -7.64) mm, rotated rx -88.46 ry -2.58 rz -120.74 deg; joints [-107.775, -126.488, -117.311, 250.645, 192.981, -175.913]
  MoveL 221 to (5.8, -27.51, -6.46) mm, rotated rx -88.2 ry -3 rz -120.93 deg; joints [-107.743, -126.316, -117.782, 251.973, 193.209, -175.334]
  MoveL 222 to (6.01, -27.06, -5.34) mm, rotated rx -88.09 ry -3.15 rz -121.19 deg; joints [-107.699, -126.095, -118.132, 252.394, 193.522, -175.21]
  MoveL 223 to (6.25, -26.58, -4.28) mm, rotated rx -88.07 ry -3.14 rz -121.56 deg; joints [-107.64, -125.829, -118.446, 252.275, 193.947, -175.371]
  MoveL 224 to (6.49, -26.1, -3.3) mm, rotated rx -88.16 ry -2.95 rz -122.06 deg; joints [-107.559, -125.51, -118.741, 251.618, 194.52, -175.815]
  MoveL 225 to (6.77, -25.58, -2.36) mm, rotated rx -88.26 ry -2.71 rz -122.71 deg; joints [-107.449, -125.141, -119.118, 250.862, 195.272, -176.337]
  MoveL 226 to (7.09, -25.02, -1.44) mm, rotated rx -88.35 ry -2.49 rz -123.51 deg; joints [-107.306, -124.733, -119.628, 250.26, 196.213, -176.822]
  MoveL 227 to (7.44, -24.43, -0.58) mm, rotated rx -88.39 ry -2.35 rz -124.45 deg; joints [-107.126, -124.306, -120.289, 249.996, 197.327, -177.189]
  MoveL 228 to (7.81, -23.83, 0.22) mm, rotated rx -88.05 ry -2.76 rz -125.23 deg; joints [-106.96, -124.059, -121.158, 251.43, 198.276, -176.859]
  MoveL 229 to (7.95, -23.62, 0.48) mm, rotated rx -87.7 ry -3.24 rz -125.33 deg; joints [-106.931, -124.115, -121.521, 252.911, 198.408, -176.338]
  Set speed (1000.0 mm/s)
  MoveL 230 to (7.95, -23.62, 0.48) mm, rotated rx -87.7 ry -3.24 rz -125.33 deg; joints [-106.931, -124.115, -121.521, 252.911, 198.408, -176.338]
  MoveL 231 to (-73.7, 33.97, -3.52) mm, rotated rx -87.7 ry -3.24 rz -125.33 deg; joints [-120.48, -124.583, -125.175, 275.69, 185.247, -157.407]
  Set speed (1000.0 mm/s)
  MoveL 232 to (-97.61, -52.9, 9.17) mm, rotated rx 116.87 ry 77.75 rz 117.4 deg; joints [-115.222, -160.521, -67.073, 59.869, 206.817, -248.045]
  MoveL 233 to (1.91, -51.05, -0.42) mm, rotated rx 116.87 ry 77.75 rz 117.4 deg; joints [-106.666, -157.292, -77.207, 72.057, 198.539, -242.335]
  MoveL 234 to (1.91, -51.05, -0.42) mm, rotated rx 116.87 ry 77.75 rz 117.4 deg; joints [-106.666, -157.292, -77.207, 72.057, 198.539, -242.335]
  Set speed (100.0 mm/s)
  MoveL 235 to (1.98, -50.31, 0.65) mm, rotated rx 145.93 ry 83.34 rz 146.1 deg; joints [-106.767, -156.936, -77.827, 72.896, 197.966, -248.957]
  MoveL 236 to (2.06, -49.53, 1.69) mm, rotated rx -132.79 ry 82.53 rz -133.03 deg; joints [-106.9, -156.676, -78.845, 72.943, 197.157, -258.807]
  MoveL 237 to (2.12, -48.9, 2.48) mm, rotated rx -105.77 ry 72.55 rz -106.49 deg; joints [-107.033, -156.424, -79.839, 73.155, 196.289, -270.577]
  MoveL 238 to (2.19, -48.24, 3.26) mm, rotated rx -98.09 ry 59.15 rz -99.4 deg; joints [-107.177, -156.189, -81.03, 73.088, 195.292, -285.261]
  MoveL 239 to (2.26, -47.54, 4.04) mm, rotated rx -94.74 ry 43.82 rz -96.83 deg; joints [-107.326, -155.977, -82.465, 72.527, 194.191, -302.405]
  MoveL 240 to (2.33, -46.83, 4.81) mm, rotated rx -92.93 ry 28.65 rz -96.09 deg; joints [-107.471, -155.776, -84.144, 71.373, 193.04, -320.158]
  MoveL 241 to (2.41, -46.1, 5.55) mm, rotated rx -91.71 ry 15.57 rz -96.34 deg; joints [-107.611, -155.543, -86.084, 69.677, 191.841, -336.538]
  MoveL 242 to (2.5, -45.3, 6.35) mm, rotated rx -90.56 ry 4.41 rz -97.24 deg; joints [-107.749, -155.223, -88.571, 66.842, 190.563, -352.592]
  MoveL 243 to (2.6, -44.41, 7.18) mm, rotated rx -89.26 ry 15.3 rz -98.39 deg; joints [-107.872, -154.712, -91.822, 62.137, 189.315, -349.039]
  MoveL 244 to (2.71, -43.5, 8) mm, rotated rx -87.64 ry 28.2 rz -98.77 deg; joints [-107.964, -153.871, -95.778, 55.147, 188.344, -346.137]
  MoveL 245 to (2.81, -42.61, 8.78) mm, rotated rx -85.29 ry 42.83 rz -97.88 deg; joints [-108.025, -152.57, -100.158, 46.187, 187.743, -343.406]
  MoveL 246 to (2.92, -41.72, 9.51) mm, rotated rx -80.79 ry 58.69 rz -94.35 deg; joints [-108.059, -150.811, -104.526, 35.894, 187.521, -340.177]
  MoveL 247 to (3.02, -40.83, 10.23) mm, rotated rx -79.22 ry 55.56 rz -94.46 deg; joints [-108.07, -148.705, -108.528, 24.799, 187.666, -356.156]
  MoveL 248 to (3.14, -39.86, 10.98) mm, rotated rx -65.59 ry 71.53 rz -81.17 deg; joints [-108.046, -146.594, -111.783, 13.72, 188.331, -351.343]
  MoveL 249 to (3.26, -38.88, 11.71) mm, rotated rx 64.56 ry -68.64 rz 98.41 deg; joints [-107.992, -144.893, -114.076, 4.417, 189.339, -183.803]
  MoveL 250 to (3.38, -37.89, 12.42) mm, rotated rx -77.64 ry -31.28 rz -112.88 deg; joints [-107.903, -143.813, -115.568, -2.522, 190.645, -113.641]
  MoveL 251 to (3.5, -36.94, 13.07) mm, rotated rx -75.71 ry -32.92 rz -115.11 deg; joints [-107.796, -143.141, -116.622, -7.575, 191.971, -121.022]
  MoveL 252 to (3.62, -35.99, 13.7) mm, rotated rx -73.75 ry -34.32 rz -117.34 deg; joints [-107.667, -142.802, -117.406, -11.238, 193.37, -126.901]
  MoveL 253 to (3.74, -35.01, 14.32) mm, rotated rx -71.78 ry -35.52 rz -119.54 deg; joints [-107.518, -142.719, -118.006, -13.79, 194.791, -131.595]
  MoveL 254 to (3.87, -34.03, 14.91) mm, rotated rx -69.83 ry -36.58 rz -121.66 deg; joints [-107.354, -142.834, -118.462, -15.441, 196.193, -135.342]
  MoveL 255 to (3.99, -33.04, 15.49) mm, rotated rx -67.9 ry -37.55 rz -123.68 deg; joints [-107.182, -143.108, -118.789, -16.338, 197.542, -138.314]
  MoveL 256 to (4.12, -32.05, 16.04) mm, rotated rx -66.16 ry -38.28 rz -125.5 deg; joints [-107.015, -143.394, -119.075, -16.924, 198.759, -140.702]
  MoveL 257 to (4.25, -31.06, 16.56) mm, rotated rx -64.37 ry -39.13 rz -127.25 deg; joints [-106.845, -143.841, -119.206, -16.834, 199.915, -142.552]
  MoveL 258 to (4.37, -30.12, 17.03) mm, rotated rx -62.98 ry -39.61 rz -128.66 deg; joints [-106.702, -144.142, -119.382, -16.905, 200.849, -144.033]
  MoveL 259 to (4.5, -29.18, 17.48) mm, rotated rx -61.57 ry -40.18 rz -130 deg; joints [-106.564, -144.53, -119.456, -16.594, 201.72, -145.21]
  MoveL 260 to (4.62, -28.23, 17.9) mm, rotated rx -59.98 ry -41 rz -131.37 deg; joints [-106.426, -145.079, -119.354, -15.715, 202.553, -146.079]
  MoveL 261 to (4.74, -27.31, 18.29) mm, rotated rx -60.23 ry -39.83 rz -131.77 deg; joints [-106.357, -144.491, -120.205, -17.902, 202.999, -147.502]
  MoveL 262 to (4.91, -25.97, 18.81) mm, rotated rx -58.36 ry -40.85 rz -133.29 deg; joints [-106.202, -145.214, -120.022, -16.473, 203.908, -148.217]
  MoveL 263 to (5.08, -24.62, 19.29) mm, rotated rx -55.73 ry -42.72 rz -135.13 deg; joints [-106.047, -146.4, -119.298, -13.605, 204.787, -148.403]
  MoveL 264 to (5.25, -23.24, 19.71) mm, rotated rx -53.13 ry -44.5 rz -136.94 deg; joints [-105.914, -147.488, -118.528, -10.901, 205.535, -148.508]
  MoveL 265 to (5.43, -21.89, 20.07) mm, rotated rx -50.85 ry -45.95 rz -138.56 deg; joints [-105.805, -148.353, -117.88, -8.72, 206.144, -148.632]
  MoveL 266 to (5.61, -20.58, 20.37) mm, rotated rx -48.96 ry -47.03 rz -139.96 deg; joints [-105.715, -149.007, -117.398, -7.073, 206.643, -148.798]
  MoveL 267 to (5.8, -19.35, 20.59) mm, rotated rx -47.63 ry -47.61 rz -141 deg; joints [-105.64, -149.408, -117.191, -6.129, 207.05, -149.068]
  MoveL 268 to (6.01, -18.15, 20.76) mm, rotated rx -46.64 ry -47.89 rz -141.85 deg; joints [-105.564, -149.673, -117.158, -5.612, 207.438, -149.442]
  MoveL 269 to (6.25, -17, 20.88) mm, rotated rx -45.77 ry -48 rz -142.65 deg; joints [-105.478, -149.888, -117.216, -5.329, 207.853, -149.918]
  MoveL 270 to (6.49, -15.91, 20.95) mm, rotated rx -45.25 ry -47.71 rz -143.27 deg; joints [-105.373, -149.967, -117.499, -5.579, 208.319, -150.6]
  MoveL 271 to (6.77, -14.83, 20.97) mm, rotated rx -44.72 ry -47.27 rz -143.97 deg; joints [-105.234, -150.043, -117.86, -6.026, 208.901, -151.464]
  MoveL 272 to (7.09, -13.76, 20.94) mm, rotated rx -44.08 ry -46.73 rz -144.82 deg; joints [-105.052, -150.158, -118.249, -6.56, 209.622, -152.493]
  MoveL 273 to (7.44, -12.71, 20.87) mm, rotated rx -43.28 ry -46.13 rz -145.82 deg; joints [-104.824, -150.335, -118.632, -7.108, 210.487, -153.656]
  MoveL 274 to (7.81, -11.72, 20.75) mm, rotated rx -41.36 ry -46.59 rz -147.4 deg; joints [-104.625, -150.955, -118.273, -6.138, 211.202, -154.262]
  MoveL 275 to (7.95, -11.39, 20.7) mm, rotated rx -39.86 ry -47.55 rz -148.36 deg; joints [-104.599, -151.448, -117.605, -4.732, 211.279, -154.044]
  Set speed (1000.0 mm/s)
  MoveL 276 to (7.95, -11.39, 20.7) mm, rotated rx -39.86 ry -47.55 rz -148.36 deg; joints [-104.599, -151.448, -117.605, -4.732, 211.279, -154.044]
  MoveL 277 to (-73.89, 13.47, -31.11) mm, rotated rx -39.86 ry -47.55 rz -148.36 deg; joints [-114.706, -162.939, -107.21, 12.795, 212.07, -134.788]

--- program Path3 (robot UR5) ---
  Smooth(1)
  Set Ref.: Frame 2 at (-32.2, -480, 32.2) mm, rotated rx 0 ry 90 rz 0 deg
  Set Tool: laser_fixture_tool
  Show laser_fixture_tool
  Set speed (1000.0 mm/s)
  MoveJ 1 to (-70.79, -56.7, 38.74) mm, rotated rx -180 ry 71.65 rz -152.9 deg; joints [-72.898, -115.526, -81.454, -103.926, 79.99, 15.417]
  MoveL 2 to (-70.79, -56.7, 38.74) mm, rotated rx -180 ry 71.65 rz -152.9 deg; joints [-72.898, -115.526, -81.454, -103.926, 79.99, 15.417]
  MoveL 3 to (13.7, -13.47, 7.25) mm, rotated rx 180 ry 71.65 rz -152.9 deg; joints [-74.585, -114.367, -96.802, -89.47, 79.126, 13.943]
  MoveL 4 to (13.7, -13.47, 7.25) mm, rotated rx 180 ry 71.65 rz -152.9 deg; joints [-74.585, -114.367, -96.802, -89.47, 79.126, 13.943]
  Set speed (100.0 mm/s)
  MoveL 5 to (13.7, -13.94, 6.31) mm, rotated rx -180 ry 73.47 rz -151.81 deg; joints [-75.503, -114.937, -95.821, -90.341, 80.672, 12.92]
  MoveL 6 to (13.7, -14.34, 5.34) mm, rotated rx -180 ry 75.36 rz -150.85 deg; joints [-76.429, -115.452, -94.939, -91.095, 82.234, 11.936]
  MoveL 7 to (13.7, -14.67, 4.34) mm, rotated rx 180 ry 77.3 rz -150.01 deg; joints [-77.36, -115.911, -94.157, -91.73, 83.807, 10.991]
  MoveL 8 to (13.7, -14.93, 3.33) mm, rotated rx 180 ry 79.28 rz -149.31 deg; joints [-78.294, -116.311, -93.48, -92.247, 85.392, 10.081]
  MoveL 9 to (13.7, -15.13, 2.3) mm, rotated rx 180 ry 81.31 rz -148.73 deg; joints [-79.231, -116.652, -92.912, -92.644, 86.984, 9.203]
  MoveL 10 to (13.7, -15.25, 1.25) mm, rotated rx -180 ry 83.36 rz -148.28 deg; joints [-80.168, -116.931, -92.453, -92.922, 88.582, 8.355]
  MoveL 11 to (13.7, -15.3, 0.21) mm, rotated rx -180 ry 85.44 rz -147.96 deg; joints [-81.103, -117.147, -92.108, -93.077, 90.184, 7.533]
  MoveL 12 to (13.7, -15.28, -0.84) mm, rotated rx 180 ry 87.53 rz -147.75 deg; joints [-82.034, -117.301, -91.878, -93.111, 91.787, 6.734]
  MoveL 13 to (13.7, -15.18, -1.89) mm, rotated rx 180 ry 89.63 rz -147.67 deg; joints [-82.961, -117.39, -91.763, -93.021, 93.39, 5.954]
  MoveL 14 to (13.7, -15.02, -2.92) mm, rotated rx 0 ry 88.27 rz 32.29 deg; joints [-83.881, -117.416, -91.766, -92.805, 94.989, 5.19]
  MoveL 15 to (13.7, -14.78, -3.95) mm, rotated rx 0 ry 86.17 rz 32.13 deg; joints [-84.792, -117.379, -91.885, -92.464, 96.583, 4.438]
  MoveL 16 to (13.7, -14.48, -4.95) mm, rotated rx 0 ry 84.09 rz 31.85 deg; joints [-85.692, -117.278, -92.121, -91.994, 98.169, 3.696]
  MoveL 17 to (13.7, -14.1, -5.93) mm, rotated rx 0 ry 82.03 rz 31.44 deg; joints [-86.581, -117.115, -92.473, -91.395, 99.745, 2.959]
  MoveL 18 to (13.7, -13.66, -6.88) mm, rotated rx 0 ry 79.99 rz 30.91 deg; joints [-87.455, -116.891, -92.939, -90.664, 101.307, 2.226]
  MoveL 19 to (13.7, -13.16, -7.8) mm, rotated rx 0 ry 77.99 rz 30.25 deg; joints [-88.314, -116.607, -93.518, -89.801, 102.853, 1.494]
  MoveL 20 to (13.7, -12.59, -8.69) mm, rotated rx 0 ry 76.03 rz 29.46 deg; joints [-89.154, -116.266, -94.207, -88.803, 104.38, 0.76]
  MoveL 21 to (13.7, -11.97, -9.53) mm, rotated rx 0 ry 74.13 rz 28.55 deg; joints [-89.975, -115.868, -95.003, -87.668, 105.884, 0.023]
  MoveL 22 to (13.7, -11.29, -10.33) mm, rotated rx 0 ry 72.28 rz 27.5 deg; joints [-90.773, -115.418, -95.903, -86.393, 107.36, -0.718]
  MoveL 23 to (13.7, -10.55, -11.08) mm, rotated rx 0 ry 70.5 rz 26.32 deg; joints [-91.547, -114.917, -96.903, -84.978, 108.806, -1.465]
  MoveL 24 to (13.7, -9.77, -11.78) mm, rotated rx 0 ry 68.8 rz 25 deg; joints [-92.294, -114.369, -97.998, -83.419, 110.217, -2.216]
  MoveL 25 to (13.7, -8.94, -12.42) mm, rotated rx 0 ry 67.18 rz 23.55 deg; joints [-93.012, -113.778, -99.184, -81.714, 111.587, -2.969]
  MoveL 26 to (13.7, -8.07, -13) mm, rotated rx 0 ry 65.66 rz 21.97 deg; joints [-93.698, -113.147, -100.457, -79.86, 112.91, -3.724]
  MoveL 27 to (13.7, -7.15, -13.52) mm, rotated rx 0 ry 64.24 rz 20.26 deg; joints [-94.35, -112.481, -101.809, -77.856, 114.182, -4.474]
  MoveL 28 to (13.7, -6.21, -13.98) mm, rotated rx 0 ry 62.94 rz 18.41 deg; joints [-94.964, -111.784, -103.237, -75.699, 115.394, -5.214]
  MoveL 29 to (13.7, -5.24, -14.37) mm, rotated rx 0 ry 61.76 rz 16.45 deg; joints [-95.538, -111.061, -104.733, -73.388, 116.54, -5.938]
  MoveL 30 to (13.7, -4.24, -14.7) mm, rotated rx 0 ry 60.72 rz 14.37 deg; joints [-96.068, -110.318, -106.292, -70.922, 117.611, -6.636]
  MoveL 31 to (13.7, -3.22, -14.96) mm, rotated rx 0 ry 59.82 rz 12.18 deg; joints [-96.55, -109.561, -107.905, -68.302, 118.599, -7.297]
  MoveL 32 to (13.7, -2.19, -15.14) mm, rotated rx 0 ry 59.06 rz 9.9 deg; joints [-96.982, -108.795, -109.565, -65.528, 119.495, -7.908]
  MoveL 33 to (13.7, -1.15, -15.26) mm, rotated rx 0 ry 58.47 rz 7.55 deg; joints [-97.359, -108.027, -111.265, -62.604, 120.288, -8.456]
  MoveL 34 to (13.7, -0.1, -15.3) mm, rotated rx 0 ry 58.03 rz 5.13 deg; joints [-97.678, -107.263, -112.997, -59.535, 120.968, -8.928]
  MoveL 35 to (13.7, 0.95, -15.27) mm, rotated rx 0 ry 57.76 rz 2.67 deg; joints [-97.933, -106.509, -114.751, -56.33, 121.524, -9.308]
  MoveL 36 to (13.7, 1.99, -15.17) mm, rotated rx 0 ry 57.67 rz 0.18 deg; joints [-98.121, -105.771, -116.518, -52.999, 121.944, -9.582]
  MoveL 37 to (13.7, 3.03, -15) mm, rotated rx 0 ry 57.74 rz -2.3 deg; joints [-98.236, -105.054, -118.29, -49.557, 122.217, -9.74]
  MoveL 38 to (13.7, 4.05, -14.75) mm, rotated rx 0 ry 57.98 rz -4.77 deg; joints [-98.274, -104.364, -120.058, -46.022, 122.331, -9.771]
  MoveL 39 to (13.7, 5.05, -14.44) mm, rotated rx 0 ry 58.39 rz -7.19 deg; joints [-98.229, -103.703, -121.812, -42.415, 122.274, -9.669]
  MoveL 40 to (13.7, 6.03, -14.06) mm, rotated rx 0 ry 58.97 rz -9.56 deg; joints [-98.098, -103.074, -123.544, -38.761, 122.037, -9.431]
  MoveL 41 to (13.7, 6.98, -13.61) mm, rotated rx 0 ry 59.7 rz -11.85 deg; joints [-97.873, -102.478, -125.246, -35.089, 121.609, -9.056]
  MoveL 42 to (13.7, 7.9, -13.1) mm, rotated rx 0 ry 60.58 rz -14.05 deg; joints [-97.55, -101.915, -126.91, -31.429, 120.982, -8.55]
  MoveL 43 to (13.7, 8.78, -12.53) mm, rotated rx 0 ry 61.6 rz -16.15 deg; joints [-97.124, -101.383, -128.53, -27.814, 120.15, -7.918]
  MoveL 44 to (13.7, 9.62, -11.9) mm, rotated rx 0 ry 62.76 rz -18.13 deg; joints [-96.59, -100.879, -130.099, -24.278, 119.106, -7.171]
  MoveL 45 to (13.7, 10.41, -11.21) mm, rotated rx 0 ry 64.05 rz -19.99 deg; joints [-95.944, -100.4, -131.613, -20.855, 117.849, -6.319]
  MoveL 46 to (13.7, 11.15, -10.47) mm, rotated rx 0 ry 65.45 rz -21.73 deg; joints [-95.182, -99.941, -133.066, -17.578, 116.376, -5.373]
  MoveL 47 to (13.7, 11.84, -9.68) mm, rotated rx 0 ry 66.95 rz -23.33 deg; joints [-94.301, -99.497, -134.455, -14.478, 114.69, -4.346]
  MoveL 48 to (13.7, 12.48, -8.85) mm, rotated rx 0 ry 68.56 rz -24.8 deg; joints [-93.299, -99.065, -135.776, -11.585, 112.796, -3.249]
  MoveL 49 to (13.7, 13.06, -7.97) mm, rotated rx 0 ry 70.25 rz -26.13 deg; joints [-92.178, -98.641, -137.023, -8.927, 110.701, -2.09]
  MoveL 50 to (13.7, 13.57, -7.06) mm, rotated rx 0 ry 72.02 rz -27.33 deg; joints [-90.939, -98.223, -138.192, -6.527, 108.414, -0.879]
  MoveL 51 to (13.7, 14.03, -6.11) mm, rotated rx 0 ry 73.85 rz -28.4 deg; joints [-89.586, -97.807, -139.279, -4.41, 105.95, 0.378]
  MoveL 52 to (13.7, 14.41, -5.14) mm, rotated rx 0 ry 75.75 rz -29.34 deg; joints [-88.127, -97.394, -140.277, -2.593, 103.325, 1.678]
  MoveL 53 to (13.7, 14.73, -4.14) mm, rotated rx 0 ry 77.7 rz -30.14 deg; joints [-86.571, -96.984, -141.182, -1.096, 100.561, 3.016]
  MoveL 54 to (13.7, 14.98, -3.12) mm, rotated rx 0 ry 79.7 rz -30.82 deg; joints [-84.932, -96.578, -141.986, 0.068, 97.68, 4.39]
  MoveL 55 to (13.7, 15.16, -2.08) mm, rotated rx 0 ry 81.73 rz -31.37 deg; joints [-83.225, -96.177, -142.682, 0.885, 94.711, 5.8]
  MoveL 56 to (13.7, 15.26, -1.04) mm, rotated rx 0 ry 83.79 rz -31.79 deg; joints [-81.47, -95.786, -143.265, 1.345, 91.682, 7.246]
  MoveL 57 to (13.7, 15.3, 0.01) mm, rotated rx 0 ry 85.87 rz -32.1 deg; joints [-79.686, -95.406, -143.728, 1.441, 88.627, 8.726]
  MoveL 58 to (13.7, 15.26, 1.06) mm, rotated rx 0 ry 87.96 rz -32.28 deg; joints [-77.898, -95.043, -144.064, 1.169, 85.579, 10.241]
  MoveL 59 to (13.7, 15.15, 2.1) mm, rotated rx -180 ry 89.94 rz 147.67 deg; joints [-76.128, -94.701, -144.269, 0.529, 82.572, 11.789]
  MoveL 60 to (13.7, 14.97, 3.14) mm, rotated rx -180 ry 87.84 rz 147.73 deg; joints [-74.399, -94.384, -144.339, -0.476, 79.641, 13.366]
  MoveL 61 to (13.7, 14.72, 4.15) mm, rotated rx -180 ry 85.74 rz 147.92 deg; joints [-72.734, -94.099, -144.27, -1.838, 76.816, 14.969]
  MoveL 62 to (13.7, 14.4, 5.15) mm, rotated rx 180 ry 83.66 rz 148.23 deg; joints [-71.153, -93.852, -144.06, -3.544, 74.128, 16.59]
  MoveL 63 to (13.7, 14.02, 6.13) mm, rotated rx -180 ry 81.61 rz 148.66 deg; joints [-69.672, -93.648, -143.708, -5.576, 71.602, 18.222]
  MoveL 64 to (13.7, 13.56, 7.08) mm, rotated rx -180 ry 79.58 rz 149.22 deg; joints [-68.306, -93.495, -143.216, -7.912, 69.26, 19.851]
  MoveL 65 to (13.7, 13.05, 7.99) mm, rotated rx -180 ry 77.59 rz 149.9 deg; joints [-67.065, -93.399, -142.584, -10.525, 67.119, 21.465]
  MoveL 66 to (13.7, 12.47, 8.86) mm, rotated rx -180 ry 75.64 rz 150.72 deg; joints [-65.957, -93.367, -141.816, -13.385, 65.193, 23.047]
  MoveL 67 to (13.7, 11.83, 9.7) mm, rotated rx 180 ry 73.74 rz 151.66 deg; joints [-64.984, -93.405, -140.916, -16.457, 63.488, 24.577]
  MoveL 68 to (13.7, 11.14, 10.49) mm, rotated rx -180 ry 71.91 rz 152.73 deg; joints [-64.148, -93.52, -139.89, -19.704, 62.01, 26.036]
  MoveL 69 to (13.7, 10.39, 11.23) mm, rotated rx 180 ry 70.15 rz 153.94 deg; joints [-63.448, -93.716, -138.744, -23.088, 60.758, 27.402]
  MoveL 70 to (13.7, 9.6, 11.91) mm, rotated rx 180 ry 68.46 rz 155.28 deg; joints [-62.879, -93.996, -137.486, -26.572, 59.73, 28.652]
  MoveL 71 to (13.7, 8.76, 12.54) mm, rotated rx -180 ry 66.86 rz 156.76 deg; joints [-62.437, -94.361, -136.125, -30.118, 58.92, 29.765]
  MoveL 72 to (13.7, 7.88, 13.11) mm, rotated rx -180 ry 65.36 rz 158.37 deg; joints [-62.116, -94.811, -134.67, -33.691, 58.319, 30.722]
  MoveL 73 to (13.7, 6.96, 13.62) mm, rotated rx 180 ry 63.97 rz 160.11 deg; joints [-61.91, -95.344, -133.132, -37.258, 57.919, 31.505]
  MoveL 74 to (13.7, 6.01, 14.07) mm, rotated rx 180 ry 62.69 rz 161.98 deg; joints [-61.811, -95.956, -131.521, -40.792, 57.708, 32.1]
  MoveL 75 to (13.7, 5.04, 14.45) mm, rotated rx -180 ry 61.54 rz 163.97 deg; joints [-61.812, -96.64, -129.848, -44.267, 57.675, 32.498]
  MoveL 76 to (13.7, 4.03, 14.76) mm, rotated rx -180 ry 60.52 rz 166.07 deg; joints [-61.906, -97.39, -128.124, -47.662, 57.806, 32.692]
  MoveL 77 to (13.7, 3.01, 15) mm, rotated rx -180 ry 59.65 rz 168.28 deg; joints [-62.086, -98.197, -126.36, -50.961, 58.091, 32.683]
  MoveL 78 to (13.7, 1.98, 15.17) mm, rotated rx 180 ry 58.93 rz 170.57 deg; joints [-62.345, -99.054, -124.566, -54.151, 58.516, 32.474]
  MoveL 79 to (13.7, 0.93, 15.27) mm, rotated rx -180 ry 58.36 rz 172.95 deg; joints [-62.678, -99.952, -122.753, -57.222, 59.069, 32.076]
  MoveL 80 to (13.7, -0.12, 15.3) mm, rotated rx -180 ry 57.96 rz 175.37 deg; joints [-63.077, -100.881, -120.928, -60.167, 59.741, 31.5]
  MoveL 81 to (13.7, -1.17, 15.25) mm, rotated rx -180 ry 57.73 rz 177.84 deg; joints [-63.538, -101.833, -119.103, -62.983, 60.518, 30.765]
  MoveL 82 to (13.7, -2.21, 15.14) mm, rotated rx -180 ry 57.67 rz -179.67 deg; joints [-64.056, -102.801, -117.285, -65.666, 61.393, 29.889]
  MoveL 83 to (13.7, -3.24, 14.95) mm, rotated rx 180 ry 57.78 rz -177.19 deg; joints [-64.624, -103.777, -115.482, -68.216, 62.354, 28.895]
  MoveL 84 to (13.7, -4.26, 14.69) mm, rotated rx 180 ry 58.05 rz -174.73 deg; joints [-65.239, -104.753, -113.701, -70.634, 63.395, 27.805]
  MoveL 85 to (13.7, -5.26, 14.37) mm, rotated rx -180 ry 58.5 rz -172.31 deg; joints [-65.896, -105.724, -111.951, -72.919, 64.506, 26.64]
  MoveL 86 to (13.7, -6.23, 13.97) mm, rotated rx -180 ry 59.1 rz -169.96 deg; joints [-66.592, -106.683, -110.236, -75.075, 65.681, 25.422]
  MoveL 87 to (13.7, -7.17, 13.51) mm, rotated rx 180 ry 59.87 rz -167.69 deg; joints [-67.322, -107.624, -108.565, -77.102, 66.914, 24.172]
  MoveL 88 to (13.7, -8.08, 12.99) mm, rotated rx 180 ry 60.78 rz -165.51 deg; joints [-68.084, -108.543, -106.942, -79.002, 68.197, 22.905]
  MoveL 89 to (13.7, -8.95, 12.41) mm, rotated rx -180 ry 61.83 rz -163.43 deg; joints [-68.874, -109.436, -105.374, -80.778, 69.527, 21.639]
  MoveL 90 to (13.7, -9.78, 11.76) mm, rotated rx -180 ry 63.02 rz -161.47 deg; joints [-69.689, -110.297, -103.867, -82.432, 70.897, 20.384]
  MoveL 91 to (13.7, -10.57, 11.07) mm, rotated rx 180 ry 64.32 rz -159.64 deg; joints [-70.526, -111.123, -102.426, -83.964, 72.305, 19.152]
  MoveL 92 to (13.7, -11.3, 10.32) mm, rotated rx 180 ry 65.75 rz -157.93 deg; joints [-71.383, -111.91, -101.055, -85.376, 73.744, 17.949]
  MoveL 93 to (13.7, -11.98, 9.52) mm, rotated rx -180 ry 67.27 rz -156.36 deg; joints [-72.257, -112.655, -99.762, -86.669, 75.213, 16.782]
  MoveL 94 to (13.7, -12.6, 8.67) mm, rotated rx 180 ry 68.9 rz -154.92 deg; joints [-73.147, -113.355, -98.549, -87.844, 76.707, 15.653]
  MoveL 95 to (13.7, -13.17, 7.79) mm, rotated rx -180 ry 72.16 rz -152.88 deg; joints [-74.732, -114.324, -96.801, -89.389, 79.554, 13.788]
  MoveL 96 to (13.7, -13.47, 7.25) mm, rotated rx 180 ry 77.69 rz -150.13 deg; joints [-77.212, -115.708, -94.418, -91.498, 84.247, 11.123]
  Set speed (1000.0 mm/s)
  MoveL 97 to (13.7, -13.47, 7.25) mm, rotated rx -180 ry 77.69 rz -150.13 deg; joints [-77.212, -115.708, -94.418, -91.498, 84.247, 11.123]
  MoveL 98 to (-71.02, -62.13, 28.57) mm, rotated rx 180 ry 77.69 rz -150.13 deg; joints [-76.335, -117.551, -78.121, -106.023, 84.707, 11.873]
